PROGRAM MAIN
VAR
	Waarde: BYTE;
	potentiometer: INT;
	nScaledMax: INT := 10;
END_VAR

(*
Potentiometer inlezen met visualisatie
Gebruik een visualisatie om de maximumwaarde en de output te tonen, alsook om de maximumwaarde te verschalen.
Rechtermuisklik op de folder VISU, selecteer 'add new' en vervolgens een VISUALISATION. Sleep vanuit de toolbox twee rectangles naar het canvas. 
Via properties window configureer je deze rectangles om de maximumwaarde nScaledMax te tonen en in te geven, en om de verschaalde output te tonen in de visu. 
*)

Waarde:=LREAL_TO_BYTE(nScaledMax*(potentiometer/32767.0));

END_PROGRAM

(* stored: Version 1.1.0.1, ProductVersion 3.1.4024.12
   POU MAIN: Id {572a745a-a627-4950-a756-b2359160babc}, SpecialFunc None *)
